(* PLC project e06cbe9c-7592-4e67-9c4f-06b90d667ec3.ecp, WAGO e!COCKPIT e!COCKPIT *)
(* stored: creationDateTime 2017-07-25T13:08:30.3259228, modificationDateTime 2017-07-25T13:03:26.2907518 *)

PROGRAM PLC_PRG

                  
                

ACTION ACT:
                      
                    
END_ACTION

METHOD METH : LTIME
                        
                      
END_METHOD
END_PROGRAM

CONFIGURATION Application
  RESOURCE Application ON PLC
    TASK PLC_Task(INTERVAL := T#10ms, PRIORITY := 14);
    PROGRAM PLC_PRG WITH PLC_Task : PLC_PRG;
  END_RESOURCE
END_CONFIGURATION
